// TIA Portal V18 export
DATA_BLOCK "Capping_Station_DB"   // DB15
VERSION : 0.1
// stored: AutoNumber true, DBAccessibleFromOPCUA true, InstanceOfName Capping_Station, InstanceOfType FB
"Capping_Station"
   // VAR_INPUT
   //    ESTOP : Bool;
   //    SerialNumber : Int;
   //    CappingOption : Int;
   //    MachineStart : Bool;
   //    CappingSensor : UInt;
   //    JogPOS : Bool;
   //    JogNEG : Bool;
   //    MoveRel : Bool;
   //    AxisXNotMoving : Bool;
   //    AxisYNotMoving : Bool;
   //    DoorSensor : Bool;
   // END_VAR
   // VAR_OUTPUT
   //    MovingUP : Bool;
   //    MovingDOWN : Bool;
   //    CSPositionUP : Bool;
   //    CSPositionDOWN : Bool;
   //    CSXYMotionLock : Bool;
   //    CappingPosition : UInt;
   //    MaintenanceNeeded : Bool;
   // END_VAR
   // VAR_IN_OUT
   //    CSMoveUP : Bool;
   //    CSMoveDOWN : Bool;
   // END_VAR
   // VAR
   //    MotionLockInternal : Bool;
   //    TimeSafety : Bool;   // Safety if the motor will keep trying to reach the position for too long
   //    SensorConversion : Real;
   //    SensorPosValMaxTrigger : UInt := 1500;
   //    SensorPosValMinTrigger : UInt := 100;
   //    ReadSensorMax : UInt;
   //    ReadSensorMin : UInt := 10000;
   //    CountSinceON : DInt;
   // END_VAR
   // VAR RETAIN
   //    CountSinceNEW : DInt;
   // END_VAR
   // VAR
   //    MaintenanceMotionLockDisabled : Bool := false;
   //    SensorPosValMin { ExternalAccessible := 'False'; ExternalVisible := 'False'; ExternalWritable := 'False'} : UInt;
   //    SensorPosValMax { ExternalAccessible := 'False'; ExternalVisible := 'False'; ExternalWritable := 'False'} : UInt;
   //    ScaleRangeMin { ExternalAccessible := 'False'; ExternalVisible := 'False'; ExternalWritable := 'False'} : UInt;
   //    ScaleRangeMax { ExternalAccessible := 'False'; ExternalVisible := 'False'; ExternalWritable := 'False'} : UInt;
   // END_VAR
BEGIN
END_DATA_BLOCK
